{attribute 'qualified_only'}
{attribute 'strict'}
TYPE E_Event :
(
	Verbose		:= 0,
	Info		:= 1,
    Warning		:= 2,
    Error		:= 3,
    Critical	:= 4
)USINT;
END_TYPE

(* stored: Version 1.1.0.1, ProductVersion 3.1.4024.12
   DUT E_Event: Id {82b5ab04-1e87-4d1a-8917-d99f26bb8a9c} *)
